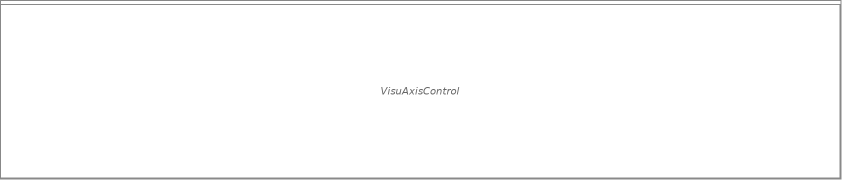
VISUALIZATION VisuAxisZ  // 842x180
    Frame (0,4 840x174)
        shows VisuAxisControl(sAxisName := sAxisZName, stAxisVisu := stAxisZ)
END_VISUALIZATION

(* stored: Version 1.1.0.1, ProductVersion 3.1.4022.6
   Visu VisuAxisZ: Id {2b2d9fdc-c630-4a86-9a21-f8968fc107fc} *)
